GLOBALCONSTANTS Hutschienenmoped_XL_strip (* Global constants *)
  (* Standard: 61499-1 *)
  (* Version 1.0, 2024-01-25, franz *)
  VAR_GLOBAL CONSTANT
    Output_strip : USINT := 0;
  END_VAR
END_GLOBALCONSTANTS
